Staubli VAL3: CmdTxtReading.pgx

program CmdTxtReading()
begin
  while true
    if nTxtTotal>2
      if bTxt1==true
        call WipeCacheRoom1()
        delay(0)

        call TxtReadRoom1()
      else
      endIf
      if bTxt2==true
        call WipeCacheRoom2()
        delay(0)

        call TxtReadRoom2()
      else
      endIf
      if bTxt3==true
        call WipeCacheRoom3()
        delay(0)

        call TxtReadRoom3()
      else
      endIf
      delay(0)
    else
    endIf
  endWhile

end
